(*

.. <legal notes>

legal notes
=================
| SPDX-FileCopyrightText: © 2025 Oleksandr Tiutyk <trofimich@gmail.com>
| SPDX-License-Identifier: LGPL-3.0-only
| For details check: LGPL-3.0-only_

.. _LGPL-3.0-only: https://www.gnu.org/licenses/lgpl-3.0.en.html

.. </legal notes>

*)

INTERFACE IMoveFromToActivityActivity EXTENDS IActivity

METHOD Configure
VAR_INPUT
	toXPosition : LREAL;
	toYPosition : LREAL;
END_VAR
END_METHOD

PROPERTY ToXPosition : LREAL
GET
END_GET
END_PROPERTY

PROPERTY ToYPosition : LREAL
GET
END_GET
END_PROPERTY

END_INTERFACE

(* stored: Version 1.1.0.1
   Itf IMoveFromToActivityActivity: Id {940fad79-65b4-4386-97b6-a2766a37107e}
   Method Configure: Id {9ccb4e38-b843-4113-be0f-07863100f907}
   Property ToXPosition: Id {d3e4c418-01c0-47cc-b47b-821dd0aa71e2}
   Get Get: Id {74ee6da6-c00d-44c9-9df5-bd2e40818b9c}
   Property ToYPosition: Id {baed957d-7c8f-4ff8-b1ad-7e58ade5f9f2}
   Get Get: Id {c4522abe-ac13-455c-ae27-fc2a0a5c360e} *)
